{attribute addProperty BoxType "EK1100-0000-0018"}
{attribute addProperty Id "Beckhoff_EJ1xxxEK1122Beckhoff_EJ1xxxEK1122_42A3763E12015A_0004_EJ1008_0000_0017EJ1008_C6161DDF9612A_0005_EJ1128_0000_0016EJ1128_C6161DDF9612A_0006_EJ1809_0000_0017EJ1809_8059E62316020A_0007_EJ1819_0000_0017EJ1819_8059E62316020A_0008_EJ1859_0000_0017EJ1859_6598BC3916020A_0009_EJ1889_0000_0017EJ1889_8059E62316020A_0003_EJ1122_0000_0016EJ1122_179A0949162"}
{attribute addProperty CRC "516160952"}
{attribute addProperty SizeInBites "968"}
{attribute addProperty SizeInBytes "121"}
TYPE Beckhoff_EJ1xxx_1EC3FDB8 EXTENDS EK1100_179A0949 :
STRUCT
	{attribute addProperty Name "Beckhoff_EJ1xxxEK1122"}
	Beckhoff_EJ1xxxEK1122 : Beckhoff_EJ1xxxEK1122_42A3763E;
	{attribute addProperty Name "A_0004_EJ1008_0000_0017"}
	A_0004_EJ1008_0000_0017 : EJ1008_C6161DDF;
	{attribute addProperty Name "A_0005_EJ1128_0000_0016"}
	A_0005_EJ1128_0000_0016 : EJ1128_C6161DDF;
	{attribute addProperty Name "A_0006_EJ1809_0000_0017"}
	A_0006_EJ1809_0000_0017 : EJ1809_8059E623;
	{attribute addProperty Name "A_0007_EJ1819_0000_0017"}
	A_0007_EJ1819_0000_0017 : EJ1819_8059E623;
	{attribute addProperty Name "A_0008_EJ1859_0000_0017"}
	A_0008_EJ1859_0000_0017 : EJ1859_6598BC39;
	{attribute addProperty Name "A_0009_EJ1889_0000_0017"}
	A_0009_EJ1889_0000_0017 : EJ1889_8059E623;
	{attribute addProperty Name "A_0003_EJ1122_0000_0016"}
	A_0003_EJ1122_0000_0016 : EJ1122_179A0949;
END_STRUCT
END_TYPE

(* stored: Version 1.2.0.0, ProductVersion 3.1.4024.9
   DUT Beckhoff_EJ1xxx_1EC3FDB8: Id {1480f91e-b347-4f18-8e57-184719cd0f33} *)
